Universal Robots URScript: happy_bday.script

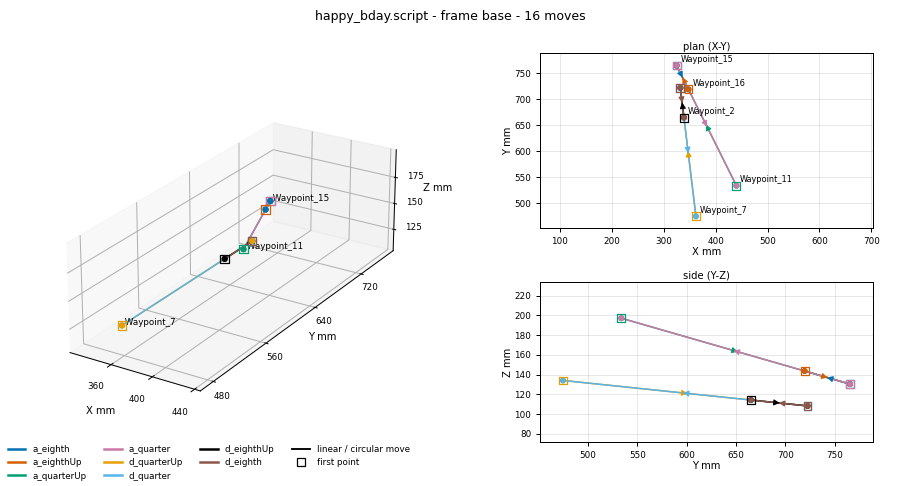
[picture p0: tool path of happy_bday.script in frame base, 16 of 16 moves have a stored position in this frame; points joined in program order, loops and branches not executed]
def happy_bday():
  global _hidden_verificationVariable=0
  set_target_payload(0.260000, [0.050000, -0.008000, 0.024000], [0.000163, 0.000163, 0.000163, 0.000000, 0.000000, 0.000000])
  set_tool_communication(False, 115200, 0, 1, 1.5, 3.5)
  set_tool_output_mode(0)
  set_tool_digital_output_mode(0, 1)
  set_tool_digital_output_mode(1, 1)
  set_tool_voltage(0)
  set_safety_mode_transition_hardness(1)
  set_tcp(p[0.028210348281514253,-0.09610723587300697,-0.09969041498611403,0.0,0.0,0.0])
  set_gravity([0.0, 0.0, 9.82])
  set_standard_analog_input_domain(0, 1)
  set_standard_analog_input_domain(1, 1)
  set_tool_analog_input_domain(0, 1)
  set_tool_analog_input_domain(1, 1)
  set_analog_outputdomain(0, 0)
  set_analog_outputdomain(1, 0)
  set_input_actions_to_default()
  global Plane_1=p[0.32571614183608727,0.7933870146316717,0.11820742021636722,-2.208244884171713,-0.24738609815952348,-1.9195085473101943]
  global Plane_2=p[0.3436052139151623,0.7478032414335104,0.10077839665899768,2.768545736097797,0.1284831553507919,1.3672805628273381]
  global Plane_3=p[0.31945151854627996,0.6757990361168175,0.09459088830114093,2.7301760593116526,-0.049483824131046385,1.4252239353300047]
  global Plane_4=p[0.3372257363094211,0.6222230974198586,0.07001667903587716,2.621672423508307,-0.12240385890263918,1.4373011913128484]
  # begin: URCap Installation Node
  #   Source: External Control, 1.0.5, FZI Research Center for Information Technology
  #   Type: External Control
  # end: URCap Installation Node
  step_count_d25caf92_c5d0_4b0d_8346_bd69edc4ae2a = 0.0
  thread Step_Counter_Thread_6b3826c6_650f_4c6e_ac5b_63da6eb62561():
    while (True):
      step_count_d25caf92_c5d0_4b0d_8346_bd69edc4ae2a = step_count_d25caf92_c5d0_4b0d_8346_bd69edc4ae2a + 1.0
      sync()
    end
  end
  run Step_Counter_Thread_6b3826c6_650f_4c6e_ac5b_63da6eb62561()
  global Waypoint_15_p=p[.324752035740, .765323943505, .130384926002, -1.494390555027, -2.277831043302, 1.156901887730]
  global Waypoint_15_q=[-2.2175437860100358, -0.2572999179838069, 0.5854005161315633, -1.0825921479197582, -1.448159388314024, -2.6781183971139746]
  global Waypoint_16_p=p[.347657429206, .719315144627, .143638713953, -1.494399401239, -2.277818707626, 1.156899707682]
  global Waypoint_16_q=[-2.2732370535480193, -0.37454839170486665, 0.7954018751726917, -1.1715508264353938, -1.4884193579303382, -2.716248337422524]
  global Waypoint_13_p=p[.347657429206, .719315144627, .143638713953, -1.494399401239, -2.277818707626, 1.156899707682]
  global Waypoint_13_q=[-2.2732370535480193, -0.37454839170486665, 0.7954018751726917, -1.1715508264353938, -1.4884193579303382, -2.716248337422524]
  global Waypoint_14_p=p[.324752035740, .765323943505, .130384926002, -1.494390555027, -2.277831043302, 1.156901887730]
  global Waypoint_14_q=[-2.2175437860100358, -0.2572999179838069, 0.5854005161315633, -1.0825921479197582, -1.448159388314024, -2.6781183971139746]
  global Waypoint_11_p=p[.439970647423, .533839164624, .197070289297, -1.494358441042, -2.277827104333, 1.156917736876]
  global Waypoint_11_q=[-2.530459845704803, -0.6687565455417506, 1.2491110730625736, -1.3336343784427385, -1.676062206371708, -2.89166459544314]
  global Waypoint_12_p=p[.324752035740, .765323943505, .130384926002, -1.494390555027, -2.277831043302, 1.156901887730]
  global Waypoint_12_q=[-2.2175437860100358, -0.2572999179838069, 0.5854005161315633, -1.0825921479197582, -1.448159388314024, -2.6781183971139746]
  global Waypoint_9_p=p[.324752035740, .765323943505, .130384926002, -1.494390555027, -2.277831043302, 1.156901887730]
  global Waypoint_9_q=[-2.2175437860100358, -0.2572999179838069, 0.5854005161315633, -1.0825921479197582, -1.448159388314024, -2.6781183971139746]
  global Waypoint_10_p=p[.439970647423, .533839164624, .197070289297, -1.494358441042, -2.277827104333, 1.156917736876]
  global Waypoint_10_q=[-2.530459845704803, -0.6687565455417506, 1.2491110730625736, -1.3336343784427385, -1.676062206371708, -2.89166459544314]
  global Waypoint_7_p=p[.362010357555, .474766328078, .134068376455, -1.613045547528, -2.136313119329, 1.151330141151]
  global Waypoint_7_q=[-2.5493923449541125, -0.7570558593208405, 1.649136843878506, -1.6208817600006542, -1.6035007246170432, -2.808236179484469]
  global Waypoint_8_p=p[.331971133677, .722315253805, .108291185217, -1.644956385011, -2.108101752441, 1.059071402778]
  global Waypoint_8_q=[-2.263843838368551, -0.37471242368731694, 0.9072483221637171, -1.3311255735209961, -1.3414958159076136, -2.600104633961813]
  global Waypoint_5_p=p[.331971133677, .722315253805, .108291185217, -1.644956385011, -2.108101752441, 1.059071402778]
  global Waypoint_5_q=[-2.263843838368551, -0.37471242368731694, 0.9072483221637171, -1.3311255735209961, -1.3414958159076136, -2.600104633961813]
  global Waypoint_6_p=p[.362010357555, .474766328078, .134068376455, -1.613045547528, -2.136313119329, 1.151330141151]
  global Waypoint_6_q=[-2.5493923449541125, -0.7570558593208405, 1.649136843878506, -1.6208817600006542, -1.6035007246170432, -2.808236179484469]
  global Waypoint_2_p=p[.338919302833, .665001489926, .114260142464, -1.637779241863, -2.114844316195, 1.080412956872]
  global Waypoint_2_q=[-2.318634812031852, -0.4877417844585352, 1.131499592457994, -1.4215563547662775, -1.3917120138751233, -2.643481318150635]
  global Waypoint_4_p=p[.331971133677, .722315253805, .108291185217, -1.644956385011, -2.108101752441, 1.059071402778]
  global Waypoint_4_q=[-2.263843838368551, -0.37471242368731694, 0.9072483221637171, -1.3311255735209961, -1.3414958159076136, -2.600104633961813]
  global Waypoint_1_p=p[.331971133677, .722315253805, .108291185217, -1.644956385011, -2.108101752441, 1.059071402778]
  global Waypoint_1_q=[-2.263843838368551, -0.37471242368731694, 0.9072483221637171, -1.3311255735209961, -1.3414958159076136, -2.600104633961813]
  global Waypoint_3_p=p[.338919302833, .665001489926, .114260142464, -1.637779241863, -2.114844316195, 1.080412956872]
  global Waypoint_3_q=[-2.318634812031852, -0.4877417844585352, 1.131499592457994, -1.4215563547662775, -1.3917120138751233, -2.643481318150635]
  def a_eighth():
    $ 31 "a_eighth" "noBreak"
    $ 32 "MoveL"
    $ 33 "Waypoint_15" "breakAfter"
    movel(pose_trans(Plane_1, pose_trans(p[-.156489454785, .686583460113, -.503627994728, 2.208244884172, .247386098160, 1.919508547310], Waypoint_15_p)), a=1.2, v=0.25)
    $ 34 "Waypoint_16" "breakAfter"
    movel(pose_trans(Plane_1, pose_trans(p[-.156489454785, .686583460113, -.503627994728, 2.208244884172, .247386098160, 1.919508547310], Waypoint_16_p)), a=1.2, v=0.25)
  end
  def a_eighthUp():
    $ 35 "a_eighthUp" "noBreak"
    $ 36 "MoveL"
    $ 37 "Waypoint_13" "breakAfter"
    movel(pose_trans(Plane_1, pose_trans(p[-.156489454785, .686583460113, -.503627994728, 2.208244884172, .247386098160, 1.919508547310], Waypoint_13_p)), a=1.2, v=0.25)
    $ 38 "Waypoint_14" "breakAfter"
    movel(pose_trans(Plane_1, pose_trans(p[-.156489454785, .686583460113, -.503627994728, 2.208244884172, .247386098160, 1.919508547310], Waypoint_14_p)), a=1.2, v=0.25)
  end
  def a_quarterUp():
    $ 39 "a_quarterUp" "noBreak"
    $ 40 "MoveL"
    $ 41 "Waypoint_11" "breakAfter"
    movel(pose_trans(Plane_1, pose_trans(p[-.156489454785, .686583460113, -.503627994728, 2.208244884172, .247386098160, 1.919508547310], Waypoint_11_p)), a=1.2, v=0.25)
    $ 42 "Waypoint_12" "breakAfter"
    movel(pose_trans(Plane_1, pose_trans(p[-.156489454785, .686583460113, -.503627994728, 2.208244884172, .247386098160, 1.919508547310], Waypoint_12_p)), a=1.2, v=0.25)
  end
  def a_quarter():
    $ 43 "a_quarter" "noBreak"
    $ 44 "MoveL"
    $ 45 "Waypoint_9" "breakAfter"
    movel(pose_trans(Plane_1, pose_trans(p[-.156489454785, .686583460113, -.503627994728, 2.208244884172, .247386098160, 1.919508547310], Waypoint_9_p)), a=1.2, v=0.25)
    $ 46 "Waypoint_10" "breakAfter"
    movel(pose_trans(Plane_1, pose_trans(p[-.156489454785, .686583460113, -.503627994728, 2.208244884172, .247386098160, 1.919508547310], Waypoint_10_p)), a=1.2, v=0.25)
  end
  def d_quarterUp():
    $ 47 "d_quarterUp" "noBreak"
    $ 48 "MoveL"
    $ 49 "Waypoint_7" "breakAfter"
    movel(pose_trans(Plane_2, pose_trans(p[-.360194635270, .718115715874, -.204939404457, -2.768545736098, -.128483155351, -1.367280562827], Waypoint_7_p)), a=1.2, v=0.25)
    $ 50 "Waypoint_8" "breakAfter"
    movel(pose_trans(Plane_2, pose_trans(p[-.360194635270, .718115715874, -.204939404457, -2.768545736098, -.128483155351, -1.367280562827], Waypoint_8_p)), a=1.2, v=0.25)
  end
  def d_quarter():
    $ 51 "d_quarter" "noBreak"
    $ 52 "MoveL"
    $ 53 "Waypoint_5" "breakAfter"
    movel(pose_trans(Plane_2, pose_trans(p[-.360194635270, .718115715874, -.204939404457, -2.768545736098, -.128483155351, -1.367280562827], Waypoint_5_p)), a=1.2, v=0.25)
    $ 54 "Waypoint_6" "breakAfter"
    movel(pose_trans(Plane_2, pose_trans(p[-.360194635270, .718115715874, -.204939404457, -2.768545736098, -.128483155351, -1.367280562827], Waypoint_6_p)), a=1.2, v=0.25)
  end
  def d_eighthUp():
    $ 55 "d_eighthUp" "noBreak"
    $ 56 "MoveL"
    $ 57 "Waypoint_2" "breakAfter"
    movel(pose_trans(Plane_2, pose_trans(p[-.360194635270, .718115715874, -.204939404457, -2.768545736098, -.128483155351, -1.367280562827], Waypoint_2_p)), a=1.2, v=0.25)
    $ 58 "Waypoint_4" "breakAfter"
    movel(pose_trans(Plane_2, pose_trans(p[-.360194635270, .718115715874, -.204939404457, -2.768545736098, -.128483155351, -1.367280562827], Waypoint_4_p)), a=1.2, v=0.25)
  end
  def d_eighth():
    $ 59 "d_eighth" "noBreak"
    $ 60 "MoveL"
    $ 61 "Waypoint_1" "breakAfter"
    movel(pose_trans(Plane_2, pose_trans(p[-.360194635270, .718115715874, -.204939404457, -2.768545736098, -.128483155351, -1.367280562827], Waypoint_1_p)), a=1.2, v=0.25)
    $ 62 "Waypoint_3" "breakAfter"
    movel(pose_trans(Plane_2, pose_trans(p[-.360194635270, .718115715874, -.204939404457, -2.768545736098, -.128483155351, -1.367280562827], Waypoint_3_p)), a=1.2, v=0.25)
  end
  while (True):
    $ 2 "Robot Program"
    $ 3 "Wait: 10.0"
    sleep(10.0)
    $ 4 "Call d_eighth"
    d_eighth()
    $ 5 "Call d_eighthUp"
    d_eighthUp()
    $ 6 "Call d_quarter"
    d_quarter()
    $ 7 "Call d_quarterUp"
    d_quarterUp()
    $ 8 "Call d_quarter"
    d_quarter()
    $ 9 "Call d_quarterUp"
    d_quarterUp()
    $ 10 "Wait: 1.0"
    sleep(1.0)
    $ 11 "Call d_eighth"
    d_eighth()
    $ 12 "Call d_eighthUp"
    d_eighthUp()
    $ 13 "Call d_quarter"
    d_quarter()
    $ 14 "Call d_quarterUp"
    d_quarterUp()
    $ 15 "Call a_quarter"
    a_quarter()
    $ 16 "Call d_quarterUp"
    d_quarterUp()
    $ 17 "Wait: 1.0"
    sleep(1.0)
    $ 18 "Call d_eighth"
    d_eighth()
    $ 19 "Call d_eighthUp"
    d_eighthUp()
    $ 20 "Call a_quarter"
    a_quarter()
    $ 21 "Call a_quarterUp"
    a_quarterUp()
    $ 22 "Call d_quarter"
    d_quarter()
    $ 23 "Call d_quarterUp"
    d_quarterUp()
    $ 24 "Call d_quarter"
    d_quarter()
    $ 25 "Call a_quarterUp"
    a_quarterUp()
    $ 26 "Call a_quarter"
    a_quarter()
    $ 27 "Call d_quarterUp"
    d_quarterUp()
    $ 28 "Call a_quarter"
    a_quarter()
    $ 29 "Call d_quarterUp"
    d_quarterUp()
    $ 30 "Wait: 2.0"
    sleep(2.0)
  end
end
